// TIA Portal project "Prrofibus" (V15.1)

(* hardware
DEVICE "HMI_1"  KTP700 Basic DP
   slot 0: "HMI_1"  KTP700 Basic DP  6AV2 123-2GA03-0AX0  15.1.0.0
   slot 1: "HMI_RT_1"  KTP700 Basic DP  6AV2 123-2GA03-0AX0  15.1.0.0
   slot 7: "HMI_1.MPI/DP_CP_1"  MPI/DP Interface  15.0.1.0
DEVICE "S71500/ET200MP station_1"  S7-1500 station
   slot 0: "Rail_0"  Rack  6ES7 590-1***0-0AA0
   slot 1: "PLC_1"  CPU 1516-3 PN/DP  6ES7 516-3AN00-0AB0  V1.8
      slot 3: "CPU display_1"  6ES7591-1BA00-0AA0
DEVICE "GSD device_1"  GSD.Device
   slot 0: "Rack_0"  Rail
   slot 0: "Slave_1"  6SE640X-1PB00-0AA0  V1.0
*)

// ===== PLC "PLC_1"  CPU 1516-3 PN/DP =====

VAR_GLOBAL   // PLC tag table "Default tag table"
   "Vel_Porcentaje" AT %MW2 : Int;
   "Vel_Deseada" AT %QW2 : Int;
   "Control_Variador" AT %QW0 : Word;
   "Vel_Real" AT %IW2 : Int;
   "Estado_Variador" AT %IW0 : Word;
   "Vel_RPM" AT %MW0 : Int;
   "Sentido_Giro" AT %M0.0 : Bool;
   "START" AT %M4.0 : Bool;
   "STOP" AT %M4.1 : Bool;
   "Motor_DER" AT %M4.2 : Bool;
   "Motor_IZQ" AT %M4.3 : Bool;
END_VAR

ORGANIZATION_BLOCK "Main"   // OB1, LAD, ProgramCycle
TITLE = "Main Program Sweep (Cycle)"
{ S7_Optimized_Access := 'TRUE' }
VERSION : 0.1
   VAR_INPUT
      Initial_Call : Bool;   // Initial call of this OB
      Remanence : Bool;   // =True, if remanent data are available
   END_VAR
BEGIN

REGION Network 1: START
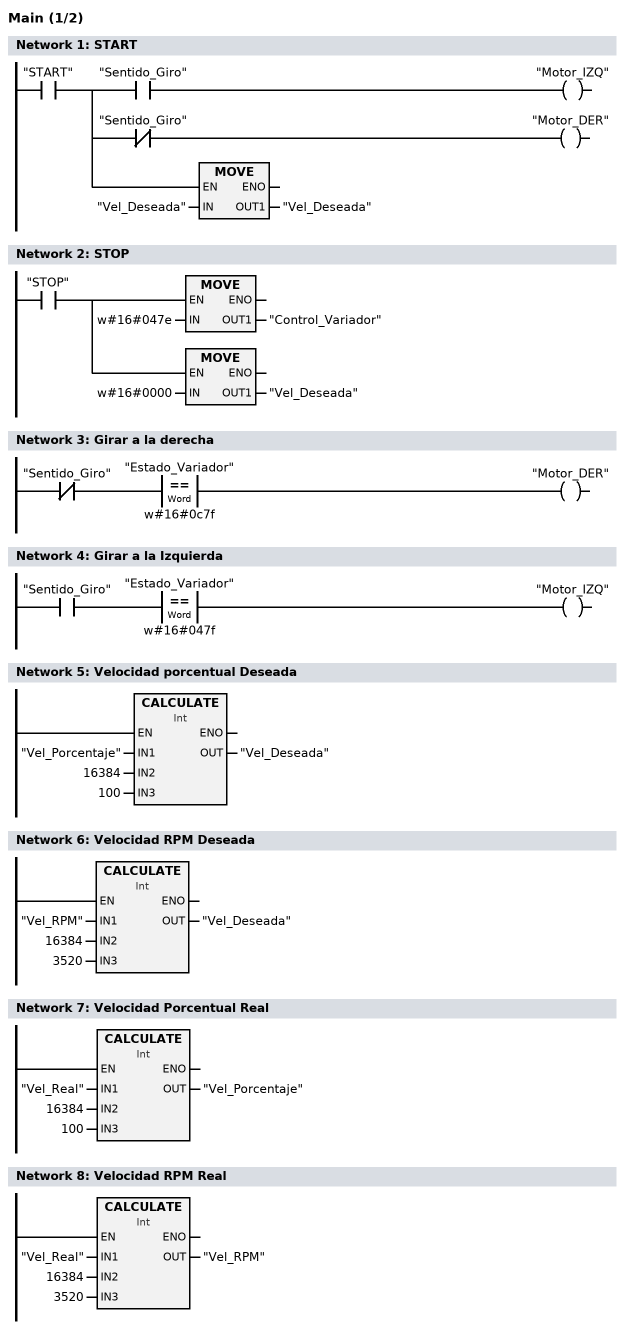
   RUNG wire#powerrail
      Contact( "START" )
      wire#w1
      Contact( "Sentido_Giro" )
      Coil( "Motor_IZQ" )
   END_RUNG
   RUNG wire#w1
      I_Contact( "Sentido_Giro" )
      Coil( "Motor_DER" )
   END_RUNG
   RUNG wire#w1
      Move(in := "Vel_Deseada", out1 => "Vel_Deseada")
   END_RUNG
   // the same network as SCL:
   "Motor_IZQ" := "START" AND "Sentido_Giro";
   "Motor_DER" := "START" AND NOT "Sentido_Giro";
   IF "START" THEN "Vel_Deseada" := "Vel_Deseada"; END_IF;
END_REGION

REGION Network 2: STOP
   RUNG wire#powerrail
      Contact( "STOP" )
      wire#w1
      Move(in := w#16#047e, out1 => "Control_Variador")
   END_RUNG
   RUNG wire#w1
      Move(in := w#16#0000, out1 => "Vel_Deseada")
   END_RUNG
   // the same network as SCL:
   IF "STOP" THEN
       "Control_Variador" := w#16#047e;
       "Vel_Deseada" := w#16#0000;
   END_IF;
END_REGION

REGION Network 3: Girar a la derecha
   RUNG wire#powerrail
      I_Contact( "Sentido_Giro" )
      { S7_Templates := "SrcType := Word" } EQ_Contact(in1 := "Estado_Variador", in2 := w#16#0c7f)
      Coil( "Motor_DER" )
   END_RUNG
   // the same network as SCL:
   "Motor_DER" := NOT "Sentido_Giro" AND ("Estado_Variador" = w#16#0c7f);
END_REGION

REGION Network 4: Girar a la Izquierda
   RUNG wire#powerrail
      Contact( "Sentido_Giro" )
      { S7_Templates := "SrcType := Word" } EQ_Contact(in1 := "Estado_Variador", in2 := w#16#047f)
      Coil( "Motor_IZQ" )
   END_RUNG
   // the same network as SCL:
   "Motor_IZQ" := "Sentido_Giro" AND ("Estado_Variador" = w#16#047f);
END_REGION

REGION Network 5: Velocidad porcentual Deseada
   RUNG wire#powerrail
      { S7_Templates := "SrcType := Int"; S7_Expression := "IN1*IN2/IN3" } Calculate(in1 := "Vel_Porcentaje", in2 := 16384, in3 := 100, out => "Vel_Deseada")
   END_RUNG
   // the same network as SCL:
   "Vel_Deseada" := "Vel_Porcentaje"*16384/100;
END_REGION

REGION Network 6: Velocidad RPM Deseada
   RUNG wire#powerrail
      { S7_Templates := "SrcType := Int"; S7_Expression := "IN1*IN2/IN3" } Calculate(in1 := "Vel_RPM", in2 := 16384, in3 := 3520, out => "Vel_Deseada")
   END_RUNG
   // the same network as SCL:
   "Vel_Deseada" := "Vel_RPM"*16384/3520;
END_REGION

REGION Network 7: Velocidad Porcentual Real
   RUNG wire#powerrail
      { S7_Templates := "SrcType := Int"; S7_Expression := "IN1*IN3/IN2" } Calculate(in1 := "Vel_Real", in2 := 16384, in3 := 100, out => "Vel_Porcentaje")
   END_RUNG
   // the same network as SCL:
   "Vel_Porcentaje" := "Vel_Real"*100/16384;
END_REGION

REGION Network 8: Velocidad RPM Real
   RUNG wire#powerrail
      { S7_Templates := "SrcType := Int"; S7_Expression := "IN1*IN3/IN2" } Calculate(in1 := "Vel_Real", in2 := 16384, in3 := 3520, out => "Vel_RPM")
   END_RUNG
   // the same network as SCL:
   "Vel_RPM" := "Vel_Real"*3520/16384;
END_REGION

REGION Network 9: Girar Motor Derecha
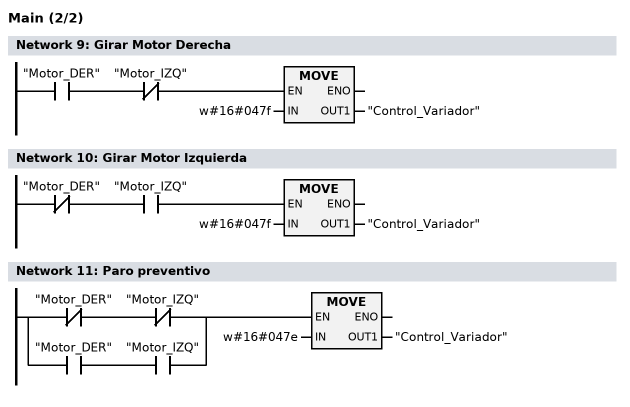
   RUNG wire#powerrail
      Contact( "Motor_DER" )
      I_Contact( "Motor_IZQ" )
      Move(in := w#16#047f, out1 => "Control_Variador")
   END_RUNG
   // the same network as SCL:
   IF "Motor_DER" AND NOT "Motor_IZQ" THEN "Control_Variador" := w#16#047f; END_IF;
END_REGION

REGION Network 10: Girar Motor Izquierda
   RUNG wire#powerrail
      I_Contact( "Motor_DER" )
      Contact( "Motor_IZQ" )
      Move(in := w#16#047f, out1 => "Control_Variador")
   END_RUNG
   // the same network as SCL:
   IF NOT "Motor_DER" AND "Motor_IZQ" THEN "Control_Variador" := w#16#047f; END_IF;
END_REGION

REGION Network 11: Paro preventivo
   RUNG wire#powerrail
      I_Contact( "Motor_DER" )
      I_Contact( "Motor_IZQ" )
      wire#w1
      Move(in := w#16#047e, out1 => "Control_Variador")
   END_RUNG
   RUNG wire#powerrail
      Contact( "Motor_DER" )
      Contact( "Motor_IZQ" )
   END_RUNG wire#w1
   // the same network as SCL:
   IF (NOT "Motor_DER" AND NOT "Motor_IZQ") OR ("Motor_DER" AND "Motor_IZQ") THEN
       "Control_Variador" := w#16#047e;
   END_IF;
END_REGION
END_ORGANIZATION_BLOCK

(* ===== HMI "HMI_RT_1" =====
system functions are stored by id; their names below are inferred from use
connection "HMI_Connection_1": IF1 B, SMART_S7_1500_OMS

HMI tags "Default tag table"
   "Tag_ScreenNumber" : UInt, internal
   "Vel_Porcentaje" : Int = PLC Vel_Porcentaje AT %MW2, 1 s
   "Vel_RPM" : Int = PLC Vel_RPM AT %MW0, 1 s
   "Sentido_Giro" : Bool = PLC Sentido_Giro AT %M0.0, 1 s
   "START" : Bool = PLC START AT %M4.0, 1 s
   "STOP" : Bool = PLC STOP AT %M4.1, 1 s

Template "Template_1" 800x480
   Button "Exit" at 714,429 size 71x50; TextOff 'Exit'; PictureOff "ExitRuntime_KTP700_Basic_DP_TR"; PictureOn "ExitRuntime_KTP700_Basic_DP_TR"
      on Release: StopRuntime(0)
   Button "Template_Button" at 614,429 size 71x50; TextOff 'Text'
   Button "Template_Button_1" at 514,429 size 71x50; TextOff 'Text'
   Button "Template_Button_2" at 414,429 size 71x50; TextOff 'Text'
   Button "Template_Button_3" at 314,429 size 71x50; TextOff 'Text'
   Button "Template_Button_4" at 214,429 size 71x50; TextOff 'Text'
   Button "Template_Button_5" at 114,429 size 71x50; TextOff 'Text'
   Button "Start screen" at 14,429 size 71x50; TextOff 'Start screen'; PictureOff "NavigateHome_KTP700_Basic_DP_TR"; PictureOn "NavigateHome_KTP700_Basic_DP_TR"
      on Release: ActivateScreen("Root screen", 0)
   SymbolicIOField "Symbolic_IO_Field_Screen" at 93,9 size 600x33; TextOff '0'; TextOn '1'; TextList "TextList_ScreenNames"
      ProcessValue <- "Tag_ScreenNumber"
      on Change: ActivateScreenByNumber("Tag_ScreenNumber", 0)
   DateTimeField "HmiScreenItemData" at 695,25 size 105x25
   DateTimeField "HmiScreenItemData_1" at 695,0 size 105x25
   GraphicView "Logo" at 0,0 size 91x51; Picture "Logo of HMI_1"

screen "Root screen" 800x480, template "Template_1"
   on GenerateScreen: SetTag("Tag_ScreenNumber", 1)
   Button "Button_1" at 173,62 size 127x49; TextOff 'Start'
      on Activate: SetBit("START")
   Button "Button_2" at 499,62 size 127x49; TextOff 'STOP'
      on Activate: SetBit("STOP")
   IOField "I/O field_1" at 255,185 size 96x32; FormatPattern 99; Unit  %
      ProcessValue <- "Vel_Porcentaje"
   IOField "I/O field_2" at 428,185 size 121x32; FormatPattern 9999; Unit  RMP
      ProcessValue <- "Vel_RPM"
   Switch "Switch_1" at 285,323 size 244x44; CaptionText 'Switch'; TextOff 'Right'; TextOn 'Left'
      ProcessValue <- "Sentido_Giro"
   TextField "Text field_1" at 277,133 size 241x43; Text 'MOTOR SPEED'
   TextField "Text field_2" at 237,269 size 347x43; Text 'SENSE OF ROTATION'
*)